# EPICS autosave request: motorApp/Db/asyn_motor_model2_settings.req
# FILE... motor_settings.req

file basic_motor_settings.req P=$(P),M=$(M)
$(P)$(M)_able.VAL
